FUNCTION_BLOCK SPLIT_SIGNED_DINT (* Teilt einen DINT-Wert in 2 einseitige Betragswerte auf: NEG_MAG = MAX(0,-Y), POS_MAG = MAX(0,Y). Sonderfall Y=DINT#-2147483648 (DINT-Minimum): -Y wuerde ueberlaufen (Zweierkomplement, |MIN| > MAX) - in diesem Fall wird NEG_MAG auf DINT#2147483647 (DINT-Maximum) begrenzt (Regelungstechnik: Saettigung statt Ueberlauf/Vorzeichenwechsel). Feuert CNF bei jedem REQ, unabhaengig von Wertaenderung - Event-Deduplizierung erfolgt aussen im Adapter-Wrapper ADI_SPLIT_SIGNED ueber je einen E_D_FF_ANY pro Seite. *)
  (* Standard: 61499-2 *)
  (* Version 1.0, 2026-09-11, Franz Höpfinger, Einfacher Value/Event-Baustein ohne Event-Dedup - wird vom Adapter-Wrapper ADI_SPLIT_SIGNED mit je einem E_D_FF_ANY pro Seite dedupliziert *)
  PACKAGE adapter::Engineering::splitting::signed;
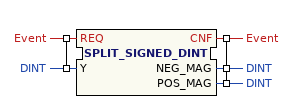
  EVENT_INPUT
    REQ WITH Y; (* Neuer Y-Wert liegt an *)
  END_EVENT
  EVENT_OUTPUT
    CNF WITH NEG_MAG, POS_MAG; (* NEG_MAG/POS_MAG berechnet *)
  END_EVENT
  VAR_INPUT
    Y : DINT; (* Eingangswert *)
  END_VAR
  VAR_OUTPUT
    NEG_MAG : DINT; (* MAX(0, -Y), bei Y=DINT#-2147483648 gesaettigt auf DINT#2147483647 *)
    POS_MAG : DINT; (* MAX(0, Y) *)
  END_VAR
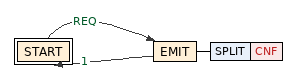
  EC_STATES
    START; (* Initial State *)
    EMIT : SPLIT -> CNF;
  END_STATES
  EC_TRANSITIONS
    START TO EMIT := REQ;
    EMIT TO START := 1;
  END_TRANSITIONS
  ALGORITHM SPLIT IN ST:
IF Y = DINT#-2147483648 THEN
	NEG_MAG := DINT#2147483647;
ELSE
	NEG_MAG := MAX(DINT#0,-Y);
END_IF;
POS_MAG := MAX(DINT#0,Y);
  END_ALGORITHM
END_FUNCTION_BLOCK
